SYSTEM TrafficLightSysAdv (* System Configuration *)
  (* Standard: 61499-1 *)
  (* Version 0.4, 2009-03-05, JHC, Holobloc Inc., Deleted Application. *)
  (* Version 0.3, 2003-12-05, JHC, Rockwell Automation, Renamed from NEWSYSTEM. *)
  (* Version 0.2, 2002-11-05, JHC, Rockwell Automation, Fixed missing (empty) FBD in Application. *)
  (* Version 0.1, 2002-01-17, JHC, Rockwell Automation, Minor cleanup *)
  (* Version 0.0, 2000-05-27, JHC, Rockwell Automation *)
  PACKAGE fb.rt.test;
  IMPORT fb.datatype.*;
  IMPORT fb.rt.*;
  IMPORT fb.rt.events.E_RESTART;
  IMPORT fb.rt.hmi.FRAME_DEVICE;
  IMPORT java.awt.*;
  DEVICE TL1_HMI : FRAME_DEVICE(BOUNDS := [0,0,300,300])
    RESOURCE HMI1 : VIEW_PANEL(SIZE := [15,15], DIA := 10)
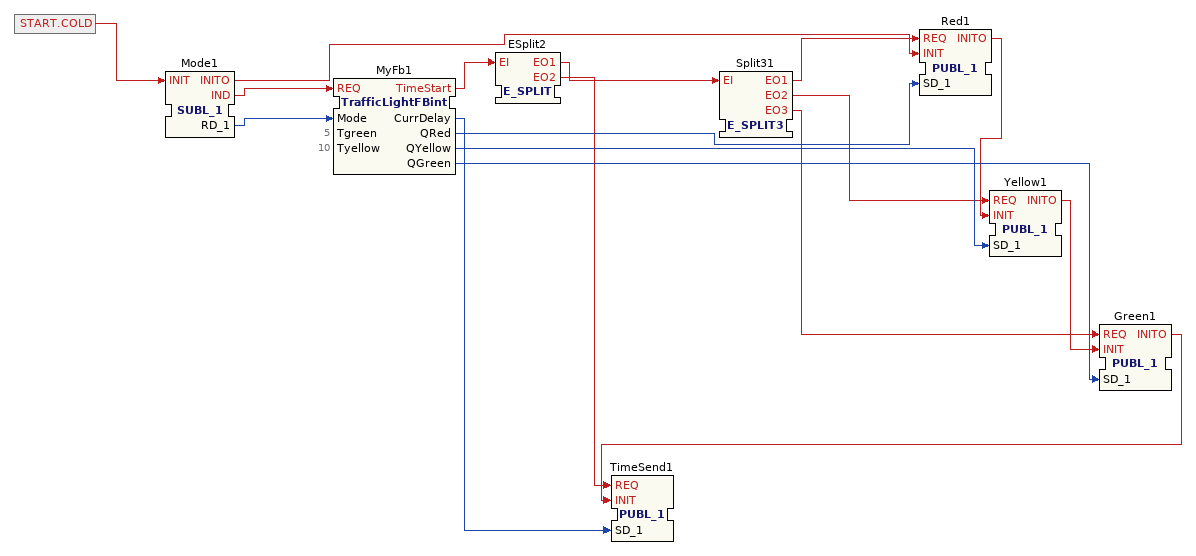
      FBS
        Red1 : PUBL_1;
        Yellow1 : PUBL_1;
        Green1 : PUBL_1;
        Split31 : E_SPLIT3;
        ESplit2 : E_SPLIT;
        TimeSend1 : PUBL_1;
        Mode1 : SUBL_1;
        MyFb1 : TrafficLightFBint(Tgreen := 5, Tyellow := 10);
      END_FBS
      EVENT_CONNECTIONS
        Split31.EO1 TO Red1.REQ;
        Split31.EO2 TO Yellow1.REQ;
        Split31.EO3 TO Green1.REQ;
        ESplit2.EO1 TO Split31.EI;
        Red1.INITO TO Yellow1.INIT;
        Yellow1.INITO TO Green1.INIT;
        ESplit2.EO2 TO TimeSend1.REQ;
        Green1.INITO TO TimeSend1.INIT;
        START.COLD TO Mode1.INIT;
        Mode1.INITO TO Red1.INIT;
        Mode1.IND TO MyFb1.REQ;
        MyFb1.TimeStart TO ESplit2.EI;
      END_CONNECTIONS
      DATA_CONNECTIONS
        MyFb1.CurrDelay TO TimeSend1.SD_1;
        Mode1.RD_1 TO MyFb1.Mode;
        MyFb1.QRed TO Red1.SD_1;
        MyFb1.QYellow TO Yellow1.SD_1;
        MyFb1.QGreen TO Green1.SD_1;
      END_CONNECTIONS
    END_RESOURCE
    RESOURCE HMI2 : VIEW_PANEL(SIZE := [15,15], DIA := 10)
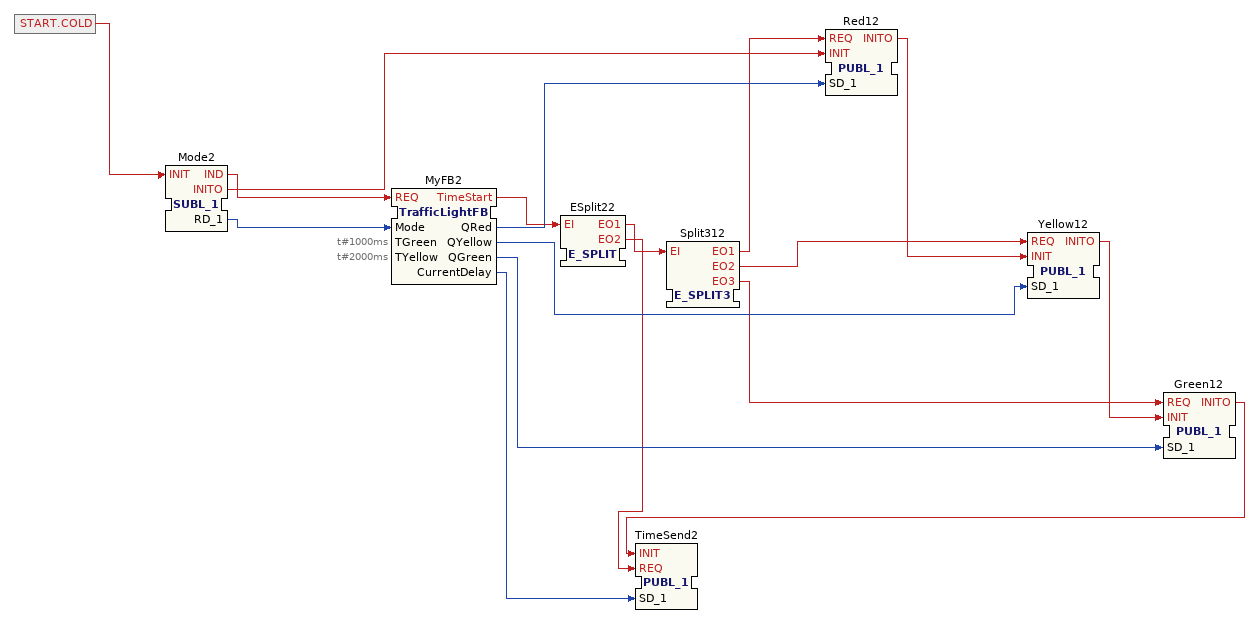
      FBS
        Red12 : PUBL_1;
        Yellow12 : PUBL_1;
        Green12 : PUBL_1;
        Split312 : E_SPLIT3;
        ESplit22 : E_SPLIT;
        MyFB2 : TrafficLightFB(TGreen := t#1000ms, TYellow := t#2000ms);
        Mode2 : SUBL_1;
        TimeSend2 : PUBL_1;
      END_FBS
      EVENT_CONNECTIONS
        Split312.EO1 TO Red12.REQ;
        Split312.EO2 TO Yellow12.REQ;
        Split312.EO3 TO Green12.REQ;
        ESplit22.EO1 TO Split312.EI;
        Red12.INITO TO Yellow12.INIT;
        Yellow12.INITO TO Green12.INIT;
        MyFB2.TimeStart TO ESplit22.EI;
        START.COLD TO Mode2.INIT;
        Mode2.IND TO MyFB2.REQ;
        Mode2.INITO TO Red12.INIT;
        Green12.INITO TO TimeSend2.INIT;
        ESplit22.EO2 TO TimeSend2.REQ;
      END_CONNECTIONS
      DATA_CONNECTIONS
        MyFB2.QRed TO Red12.SD_1;
        MyFB2.QYellow TO Yellow12.SD_1;
        MyFB2.QGreen TO Green12.SD_1;
        Mode2.RD_1 TO MyFB2.Mode;
        MyFB2.CurrentDelay TO TimeSend2.SD_1;
      END_CONNECTIONS
    END_RESOURCE
  END_DEVICE
  DEVICE Controller : FRAME_DEVICE(BOUNDS := [300,0,300,300])
    RESOURCE Ctrl1 : VIEW_PANEL(DIA := 10, SIZE := [15,15])
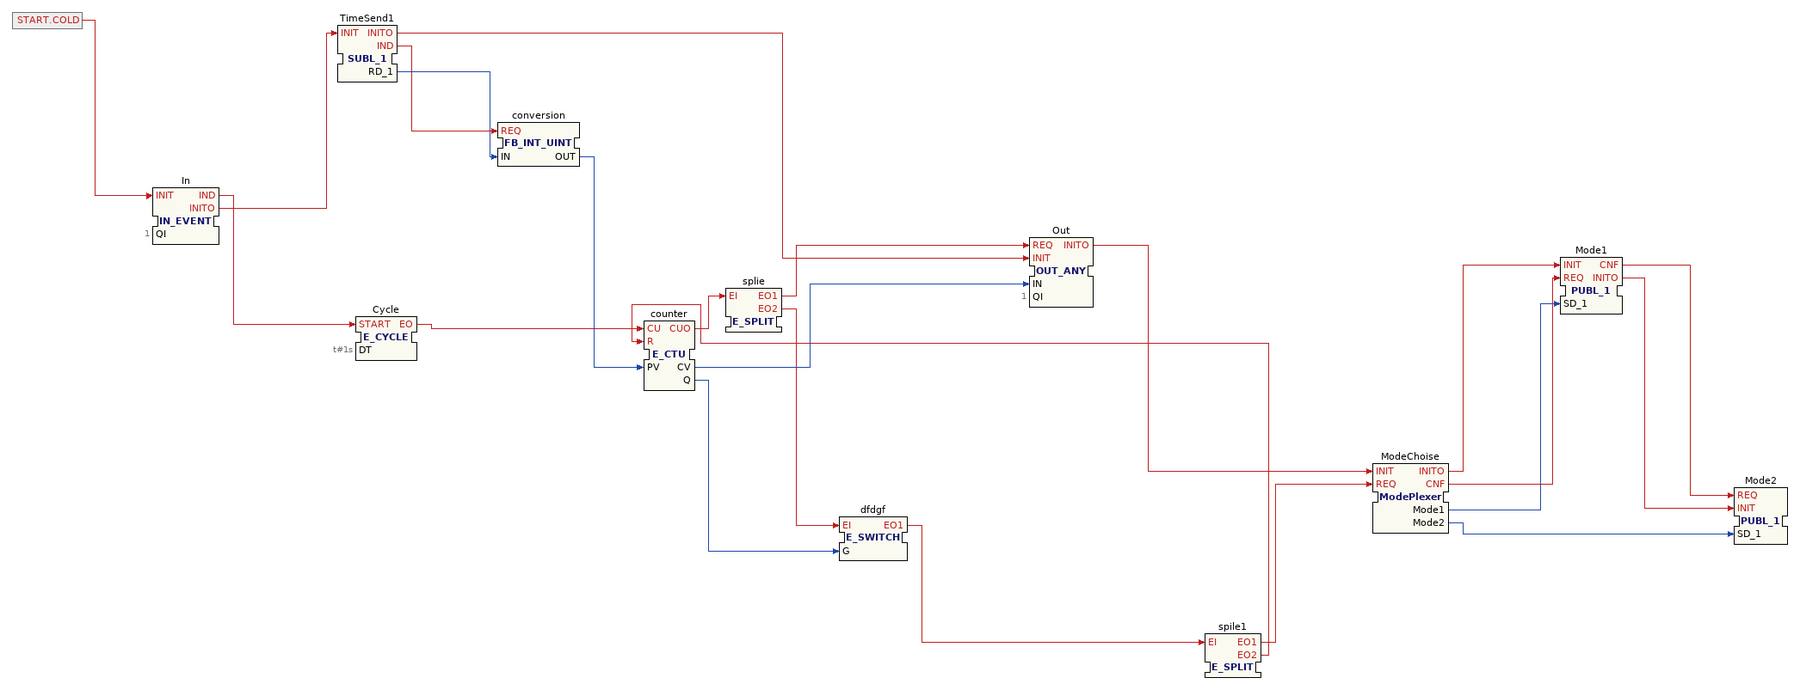
      FBS
        ModeChoise : ModePlexer;
        Cycle : E_CYCLE(DT := t#1s);
        In : IN_EVENT(QI := 1);
        Out : OUT_ANY(QI := 1);
        counter : E_CTU;
        dfdgf : E_SWITCH;
        splie : E_SPLIT;
        spile1 : E_SPLIT;
        Mode1 : PUBL_1;
        Mode2 : PUBL_1;
        TimeSend1 : SUBL_1;
        conversion : FB_INT_UINT;
      END_FBS
      EVENT_CONNECTIONS
        START.COLD TO In.INIT;
        In.IND TO Cycle.START;
        Cycle.EO TO counter.CU;
        Out.INITO TO ModeChoise.INIT;
        counter.CUO TO splie.EI;
        splie.EO1 TO Out.REQ;
        splie.EO2 TO dfdgf.EI;
        dfdgf.EO1 TO spile1.EI;
        spile1.EO1 TO ModeChoise.REQ;
        spile1.EO2 TO counter.R;
        ModeChoise.INITO TO Mode1.INIT;
        ModeChoise.CNF TO Mode1.REQ;
        Mode1.CNF TO Mode2.REQ;
        Mode1.INITO TO Mode2.INIT;
        In.INITO TO TimeSend1.INIT;
        TimeSend1.INITO TO Out.INIT;
        TimeSend1.IND TO conversion.REQ;
      END_CONNECTIONS
      DATA_CONNECTIONS
        counter.CV TO Out.IN;
        counter.Q TO dfdgf.G;
        ModeChoise.Mode1 TO Mode1.SD_1;
        ModeChoise.Mode2 TO Mode2.SD_1;
        TimeSend1.RD_1 TO conversion.IN;
        conversion.OUT TO counter.PV;
      END_CONNECTIONS
    END_RESOURCE
  END_DEVICE
  DEVICE VIew : FRAME_DEVICE(BOUNDS := [600,0,300,300])
    RESOURCE TL1_View : VIEW_PANEL(DIA := 10, SIZE := [30,30])
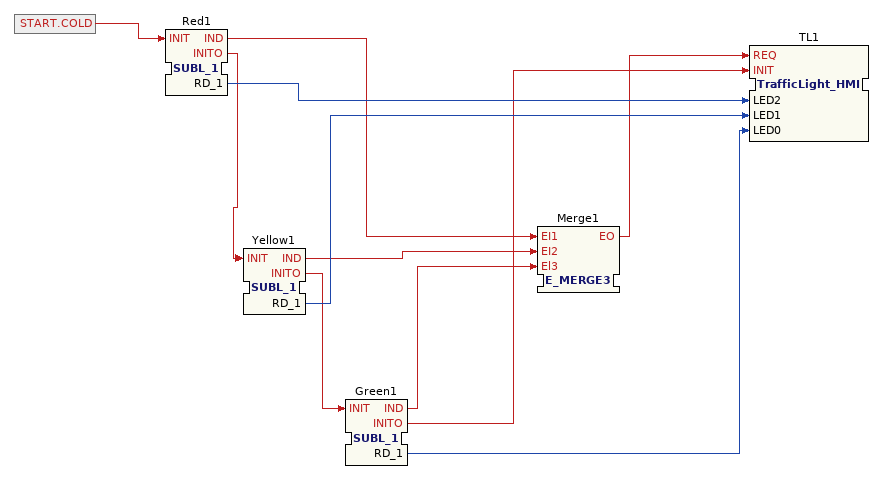
      FBS
        Red1 : SUBL_1;
        TL1 : TrafficLight_HMI;
        Yellow1 : SUBL_1;
        Green1 : SUBL_1;
        Merge1 : E_MERGE3;
      END_FBS
      EVENT_CONNECTIONS
        Red1.IND TO Merge1.EI1;
        Yellow1.IND TO Merge1.EI2;
        Green1.IND TO Merge1.El3;
        Merge1.EO TO TL1.REQ;
        START.COLD TO Red1.INIT;
        Red1.INITO TO Yellow1.INIT;
        Yellow1.INITO TO Green1.INIT;
        Green1.INITO TO TL1.INIT;
      END_CONNECTIONS
      DATA_CONNECTIONS
        Red1.RD_1 TO TL1.LED2;
        Yellow1.RD_1 TO TL1.LED1;
        Green1.RD_1 TO TL1.LED0;
      END_CONNECTIONS
    END_RESOURCE
    RESOURCE TL2_View : VIEW_PANEL(DIA := 10, SIZE := [30,30])
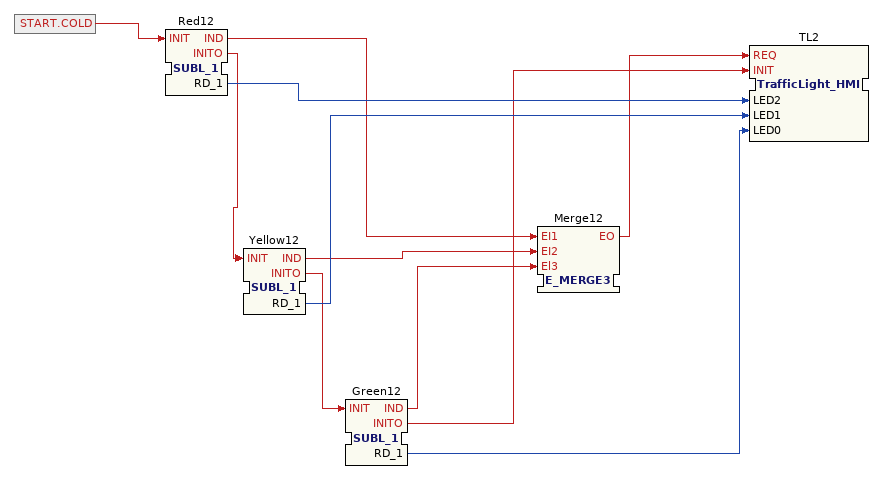
      FBS
        Red12 : SUBL_1;
        TL2 : TrafficLight_HMI;
        Yellow12 : SUBL_1;
        Green12 : SUBL_1;
        Merge12 : E_MERGE3;
      END_FBS
      EVENT_CONNECTIONS
        Red12.IND TO Merge12.EI1;
        Yellow12.IND TO Merge12.EI2;
        Green12.IND TO Merge12.El3;
        Merge12.EO TO TL2.REQ;
        START.COLD TO Red12.INIT;
        Red12.INITO TO Yellow12.INIT;
        Yellow12.INITO TO Green12.INIT;
        Green12.INITO TO TL2.INIT;
      END_CONNECTIONS
      DATA_CONNECTIONS
        Red12.RD_1 TO TL2.LED2;
        Yellow12.RD_1 TO TL2.LED1;
        Green12.RD_1 TO TL2.LED0;
      END_CONNECTIONS
    END_RESOURCE
  END_DEVICE
END_SYSTEM
